FUNCTION_BLOCK fb_ArmBasketRotateCtrl
VAR_INPUT
	bEn 							: BOOL;
	bStart			 			: BOOL;
	bRotateBasketRS_Cw			: BOOL;
	bRotateBasketRS_Ccw		: BOOL;
	bRotateBasketRS_Lock		: BOOL;
	bRotateBasketRS_Unlock		: BOOL;
	bDeactivatedMode 			: BOOL;
	iRotateBasketDelayTimeSV	: INT;
END_VAR
VAR_OUTPUT
	bRotateBasketAV_Cw			: BOOL;
	bRotateBasketAV_Ccw		: BOOL;
	bRotateBasketAV_Lock		: BOOL;
	bRotateBasketAV_Unlock		: BOOL;

END_VAR
VAR

	bStep1: BOOL;
	bStep2: BOOL;
	tRotateBasketDelay: TON;
END_VAR

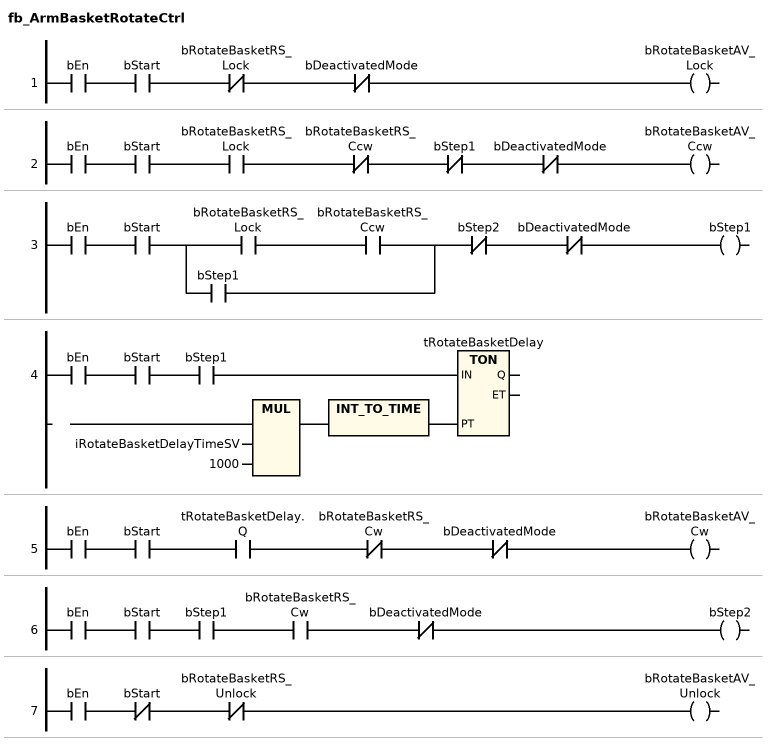
// NETWORK 1
bRotateBasketAV_Lock := bEn AND bStart AND NOT bRotateBasketRS_Lock AND NOT bDeactivatedMode;

// NETWORK 2
bRotateBasketAV_Ccw := bEn AND bStart AND bRotateBasketRS_Lock AND NOT bRotateBasketRS_Ccw AND NOT bStep1 AND NOT bDeactivatedMode;

// NETWORK 3
bStep1 := (bEn AND bStart AND (bRotateBasketRS_Lock AND bRotateBasketRS_Ccw OR bStep1)) AND NOT bStep2 AND NOT bDeactivatedMode;

// NETWORK 4
tRotateBasketDelay(IN := bEn AND bStart AND bStep1, PT := INT_TO_TIME(iRotateBasketDelayTimeSV * 1000)); // TON

// NETWORK 5
bRotateBasketAV_Cw := bEn AND bStart AND tRotateBasketDelay.Q AND NOT bRotateBasketRS_Cw AND NOT bDeactivatedMode;

// NETWORK 6
bStep2 := bEn AND bStart AND bStep1 AND bRotateBasketRS_Cw AND NOT bDeactivatedMode;

// NETWORK 7
bRotateBasketAV_Unlock := bEn AND NOT bStart AND NOT bRotateBasketRS_Unlock;

END_FUNCTION_BLOCK

(* stored: Version 1.1.0.1, ProductVersion 3.1.4024.12
   POU fb_ArmBasketRotateCtrl: Id {0272dddd-e7e5-4ece-b7b1-43ac288b896a}, SpecialFunc None *)
